(* IEC 61131-3 sources: com.logicals.lc3.webinar/usRTS_RPMControl_iSOC/src_FB_LIB_SAFE/Numeric/UDINT, 8 files *)

(* ---- wADD_UDINT_2.iecst ---- *)
NAMESPACE logicals.web.standard
NAMESPACE numeric

/*
 * Function block wrapper for IEC 61131-3 ADD<br>
 * IN1 =  1st value (UDINT)<br>
 * IN2 =  2nd value (UDINT)<br>
 * OUT = Sum of all input values (UDINT)<br>
 */
FUNCTION_BLOCK wADD_UDINT_2
	{ vNameAlignment:="center"; altName:="+"; bgColor:="Plum"; width:=40; hideIONames; }
	VAR_INPUT
		IN1 : UDINT;
		IN2 : UDINT;
	END_VAR
	VAR_OUTPUT
		OUT : UDINT;
	END_VAR

	OUT := ADD(IN1:=IN1, IN2:=IN2, ENO=>ENO);
END_FUNCTION_BLOCK

END_NAMESPACE
END_NAMESPACE

(* ---- wADD_UDINT_3.iecst ---- *)
NAMESPACE logicals.web.standard
NAMESPACE numeric

/*
 * Function block wrapper for IEC 61131-3 ADD<br>
 * IN1 =  1st value (UDINT)<br>
 * IN2 =  2nd value (UDINT)<br>
 * IN3 =  3rd value (UDINT)<br>
 * OUT = Sum of all input values (UDINT)<br>
 */
FUNCTION_BLOCK wADD_UDINT_3
	{ vNameAlignment:="center"; altName:="+"; bgColor:="Plum"; width:=40; hideIONames; }
	VAR_INPUT
		IN1 : UDINT;
		IN2 : UDINT;
		IN3 : UDINT;
	END_VAR
	VAR_OUTPUT
		OUT : UDINT;
	END_VAR

	OUT := ADD(IN1:=IN1, IN2:=IN2, IN3:=IN3, ENO=>ENO);
END_FUNCTION_BLOCK

END_NAMESPACE
END_NAMESPACE

(* ---- wADD_UDINT_4.iecst ---- *)
NAMESPACE logicals.web.standard
NAMESPACE numeric

/*
 * Function block wrapper for IEC 61131-3 ADD<br>
 * IN1 =  1st value (UDINT)<br>
 * IN2 =  2nd value (UDINT)<br>
 * IN3 =  3rd value (UDINT)<br>
 * IN4 =  4th value (UDINT)<br>
 * OUT = Sum of all input values (UDINT)<br>
 */
FUNCTION_BLOCK wADD_UDINT_4
	{ vNameAlignment:="center"; altName:="+"; bgColor:="Plum"; width:=40; hideIONames; }
	VAR_INPUT
		IN1 : UDINT;
		IN2 : UDINT;
		IN3 : UDINT;
		IN4 : UDINT;
	END_VAR
	VAR_OUTPUT
		OUT : UDINT;
	END_VAR

	OUT := ADD(IN1:=IN1, IN2:=IN2, IN3:=IN3, IN4:=IN4, ENO=>ENO);
END_FUNCTION_BLOCK

END_NAMESPACE
END_NAMESPACE

(* ---- wDIV_UDINT.iecst ---- *)
NAMESPACE logicals.web.standard
NAMESPACE numeric

/*
 * Function block wrapper for IEC 61131-3 DIV<br>
 * IN1 =  1st value (UDINT)<br>
 * IN2 =  2nd value (UDINT)<br>
 * OUT = quotient of IN1 divided by IN2 (UDINT)<br>
 */
FUNCTION_BLOCK wDIV_UDINT
	{ vNameAlignment:="center"; altName:="/"; bgColor:="Plum"; width:=40; hideIONames; }
	VAR_INPUT
		IN1 : UDINT;
		IN2 : UDINT;
	END_VAR
	VAR_OUTPUT
		OUT : UDINT;
	END_VAR

	OUT := DIV(IN1:=IN1, IN2:=IN2, ENO=>ENO);
END_FUNCTION_BLOCK

END_NAMESPACE
END_NAMESPACE

(* ---- wMUL_UDINT_2.iecst ---- *)
NAMESPACE logicals.web.standard
NAMESPACE numeric

/*
 * Function block wrapper for IEC 61131-3 MUL<br>
 * IN1 =  1st value (UDINT)<br>
 * IN2 =  2nd value (UDINT)<br>
 * OUT = Product of multiplication of all inputs (UDINT)<br>
 */
FUNCTION_BLOCK wMUL_UDINT_2
	{ vNameAlignment:="center"; altName:="*"; bgColor:="Plum"; width:=40; hideIONames; }
	VAR_INPUT
		IN1 : UDINT;
		IN2 : UDINT;
	END_VAR
	VAR_OUTPUT
		OUT : UDINT;
	END_VAR

	OUT := MUL(IN1:=IN1, IN2:=IN2, ENO=>ENO);
END_FUNCTION_BLOCK

END_NAMESPACE
END_NAMESPACE

(* ---- wMUL_UDINT_3.iecst ---- *)
NAMESPACE logicals.web.standard
NAMESPACE numeric

/*
 * Function block wrapper for IEC 61131-3 MUL<br>
 * IN1 =  1st value (UDINT)<br>
 * IN2 =  2nd value (UDINT)<br>
 * IN3 =  3rd value (UDINT)<br>
 * OUT = Product of multiplication of all inputs (UDINT)<br>
 */
FUNCTION_BLOCK wMUL_UDINT_3
	{ vNameAlignment:="center"; altName:="*"; bgColor:="Plum"; width:=40; hideIONames; }
	VAR_INPUT
		IN1 : UDINT;
		IN2 : UDINT;
		IN3 : UDINT;
	END_VAR
	VAR_OUTPUT
		OUT : UDINT;
	END_VAR

	OUT := MUL(IN1:=IN1, IN2:=IN2, IN3:=IN3, ENO=>ENO);
END_FUNCTION_BLOCK

END_NAMESPACE
END_NAMESPACE

(* ---- wMUL_UDINT_4.iecst ---- *)
NAMESPACE logicals.web.standard
NAMESPACE numeric

/*
 * Function block wrapper for IEC 61131-3 MUL<br>
 * IN1 =  1st value (UDINT)<br>
 * IN2 =  2nd value (UDINT)<br>
 * IN3 =  3rd value (UDINT)<br>
 * IN4 =  4th value (UDINT)<br>
 * OUT = Product of multiplication of all inputs (UDINT)<br>
 */
FUNCTION_BLOCK wMUL_UDINT_4
	{ vNameAlignment:="center"; altName:="*"; bgColor:="Plum"; width:=40; hideIONames; }
	VAR_INPUT
		IN1 : UDINT;
		IN2 : UDINT;
		IN3 : UDINT;
		IN4 : UDINT;
	END_VAR
	VAR_OUTPUT
		OUT : UDINT;
	END_VAR

	OUT := MUL(IN1:=IN1, IN2:=IN2, IN3:=IN3, IN4:=IN4, ENO=>ENO);
END_FUNCTION_BLOCK

END_NAMESPACE
END_NAMESPACE

(* ---- wSUB_UDINT.iecst ---- *)
NAMESPACE logicals.web.standard
NAMESPACE numeric

/*
 * Function block wrapper for IEC 61131-3 SUB<br>
 * IN1 =  1st value (UDINT)<br>
 * IN2 =  2nd value (UDINT)<br>
 * OUT = IN1 minus IN2 (UDINT)<br>
 */
FUNCTION_BLOCK wSUB_UDINT
	{ vNameAlignment:="center"; altName:="-"; bgColor:="Plum"; width:=40; hideIONames; }
	VAR_INPUT
		IN1 : UDINT;
		IN2 : UDINT;
	END_VAR
	VAR_OUTPUT
		OUT : UDINT;
	END_VAR

	OUT := SUB(IN1:=IN1, IN2:=IN2, ENO=>ENO);
END_FUNCTION_BLOCK

END_NAMESPACE
END_NAMESPACE
